(* CoDeSys 2.3.9.47 project: clv-199-wg-001.pro *)
(* Author: Diego Bernini *)
(* Libraries: SerComm.lib 31.5.11 08:54:36, SysLibEvent.lib 2.12.10 14:48:34, SysLibFile.lib 2.12.10 14:48:34, SysLibPlcCtrl.lib 2.12.10 14:48:32, SysLibRtc.lib 2.12.10 14:48:32, SysLibSockets.lib 10.2.11 09:20:54, 01_Lib_ClevergyUtils\ClevergyUtils_wg880_v2.lib 27.7.16 09:27:07, Util.lib 26.9.14 11:12:46, Visual.lib 2.12.10 14:48:34, WagoLibIdent.lib 25.2.13 11:12:16, WagoLibStatus.lib 2.12.10 14:48:32, Standard.lib 2.12.10 14:48:34, SYSLIBCALLBACK.LIB 2.12.10 14:48:32, mod_com.lib 2.12.10 14:48:32, MBus_03.lib 9.2.13 17:51:58, Modb_l05.lib 13.5.15 10:30:08, Serial_Interface_01.lib 22.4.13 12:50:14, WagoLibMBX_01.lib 20.3.12 16:32:40, WagoLibModbus_IP_01.lib 24.7.13 15:05:58, SysLibTime.lib 2.12.10 14:48:32 *)

(* PLC configuration (modules and I/O channels)
0750-1506 8DI / 8DO 24V DC 0.5A [Type_34_8_Channels] node 0, in %IB20 out %QB20 {INTTypePAAssignment = PLC; INTTypeModule = plugged}
  OUT2_VPN AT %IX10.0 [BOOLOnX_I] Ch_1 Digital input
  LAMP_AL AT %QX10.0 [BOOLOnX_Q] Ch_1 Digital output
  STATO_PORTA_QE AT %IX10.1 [BOOLOnX_I] Ch_2 Digital input
  AT %QX10.1 [BOOLOnX_Q] Ch_2 Digital output
  AT %IX10.2 [BOOLOnX_I] Ch_3 Digital input
  AT %QX10.2 [BOOLOnX_Q] Ch_3 Digital output
  AT %IX10.3 [BOOLOnX_I] Ch_4 Digital input
  AT %QX10.3 [BOOLOnX_Q] Ch_4 Digital output
  AT %IX10.4 [BOOLOnX_I] Ch_5 Digital input
  AT %QX10.4 [BOOLOnX_Q] Ch_5 Digital output
  AT %IX10.5 [BOOLOnX_I] Ch_6 Digital input
  AT %QX10.5 [BOOLOnX_Q] Ch_6 Digital output
  AT %IX10.6 [BOOLOnX_I] Ch_7 Digital input
  AT %QX10.6 [BOOLOnX_Q] Ch_7 Digital output
  AT %IX10.7 [BOOLOnX_I] Ch_8 Digital input
  AT %QX10.7 [BOOLOnX_Q] Ch_8 Digital output
AT %IB0 [BYTEOnB_I] First Byte of 8
AT %QB0 [BYTEOnB_Q] First Byte of 8
AT %IB8 [BYTEOnB_I] First Byte of 8
AT %QB8 [BYTEOnB_Q] First Byte of 8
0750-0650/0003-0000#03 RS 232 C Interface (Adjustable), 3 Byte [Type_21_1_Channels] node 3, in %IB24 out %QB24 {INTTypePAAssignment = PLC; INTTypeModule = plugged}
  AT %IX8.0 [BOOLOnX_I] Transmission acknowledgement
  AT %IX8.1 [BOOLOnX_I] Reception request
  AT %IX8.2 [BOOLOnX_I] Initialization acknowledgement
  AT %IX8.3 [BOOLOnX_I] Input buffer is full
  AT %IX8.4 [BOOLOnX_I] Number of received characters Bit 0
  AT %IX8.5 [BOOLOnX_I] Number of received characters Bit 1
  AT %IX8.6 [BOOLOnX_I] Number of received characters Bit 2
  AT %IB17 [BYTEOnB_I] Input data Byte 0
  AT %IB18 [BYTEOnB_I] Input data Byte 1
  AT %IB19 [BYTEOnB_I] Input data Byte 2
  AT %QX8.0 [BOOLOnX_Q] Transmission request
  AT %QX8.1 [BOOLOnX_Q] Reception acknowledgement
  AT %QX8.2 [BOOLOnX_Q] Initialization request
  AT %QX8.4 [BOOLOnX_Q] Number of characters Bit 0
  AT %QX8.5 [BOOLOnX_Q] Number of characters Bit 1
  AT %QX8.6 [BOOLOnX_Q] Number of characters Bit 2
  AT %QB17 [BYTEOnB_Q] Output data Byte 0
  AT %QB18 [BYTEOnB_Q] Output data Byte 1
  AT %QB19 [BYTEOnB_Q] Output data Byte 2
Fieldbus variables [FB_VARS] node 1, in %IB0 out %QB0
Flag variables [FLAG_VARS] node 2, in %IB0 out %QB0
Modbus-Master [MB_MASTER] node 3, in %IB0 out %QB0
*)

(* Global variable list: Global_Constants *)
VAR_GLOBAL CONSTANT

	Plant_NAME		: STRING :='cySN:199  cyVER:0 - Humanitas PIO X ';
	Plant_SN			: DWORD  :=199;  	         	(* S/N Impianto di telecontrollo *)
	Plant_SW_VER		: WORD   :=0;				(* Versione SW installata *)

	(* Plant-dependent constants *)
	(*Plant_ANZ_Frer			: BYTE	 :=24; *)
	Plant_ANZ_ABB		: BYTE	 :=19;
	(*Plant_GASM			: BYTE	 :=1; *)

	MODBUS_MAX_DEVICE	:BYTE:=19;
	MODBUS_MAX_REG 		: BYTE:=10;
	POLLING_TIME				:TIME:=T#10s;

	(* Filesystem *)
	FilesPath  		: STRING :='S:\';

	(* TCP Logger *)
	Logger_SERVER		: STRING:='';
	Logger_IP				: STRING:='192.168.100.3';
	Logger_PORT			: WORD  :=80;
	Logger_GETSTART		: STRING:='GET /cygmsrv/hsgm.ashx?';
	Logger_GETEND		: STRING:='$R$N$R$N';
	Logger_CHECK			: STRING:='True';
	Logger_CRLF			: STRING:='$R$N';
	Logger_DataFile			: STRING:='S:\LOG.DAT';
	Logger_DataFileOld		: STRING:='S:\LOG.BCK';
	Logger_IndexFile		: STRING:='S:\LOG.IDX';
	Logger_ConnRetries		: BYTE:=5;
	Logger_RecoverMsgs	: BYTE:=25;

	(* TCP Remote *)
	Remote_PORT			: WORD  :=10;
	Remote_WELCOME	: STRING:='Connected$R$N';
	Remote_OK				: STRING:='OK$R$N';
	Remote_ERROR		: STRING:='ERROR$R$N';

	(* TCP Sockets *)
	MAX_SEND_TCP_SERVER					 : DWORD:=6000;(*60000*)
	MAX_RECEIVE_TCP_SERVER				 : DWORD:=3000;
	MAX_RECEIVE_TCP_SERVER_SOCKET	  : DWORD:=1500;
	MAX_SEND_TCP_CLIENT					 : DWORD:=6000;(*15000*)
	MAX_RECEIVE_TCP_CLIENT				 : DWORD:=1500;
	MAX_RECEIVE_TCP_CLIENT_SOCKET		 : DWORD:=1500;
	MAX_RECEIVE_UDP_SERVER				 : INT  :=1472;
	MAX_RECEIVE_UDP_CLIENT				 : INT  :=1472;
	CONNECT_WATCHDOG_TIME				 : TIME :=t#10s;

	(* Colour defines *)
	COLOR_RED			: DWORD	:= 16#2020F0;
	COLOR_YELLOW		: DWORD	:= 16#20F0F0;
	COLOR_GREEN			: DWORD	:= 16#20F020;
	COLOR_GREEN_OFF		: DWORD := 16#006000;

END_VAR

(* Global variable list: Global_Variables *)
VAR_GLOBAL

	SYS    : typ_SYS;
	Logger : typ_Logger;

	Lamp	:	LAMP_AL_GENERALE; (* Per gestione allarme generico impianto *)

	MODB01 : obj_MODBUS	:= ( ID:=1 , (*COM:=2,*) BAUDRATE:=BAUD_9600, RS485:=TRUE, STOP_BITS:=STOPBITS_2,TIME_OUT_TIME:=t#1s);
	MODB02 : obj_MODBUS	:= ( ID:=2 , (*COM:=3,*) BAUDRATE:=BAUD_9600, RS485:=TRUE, STOP_BITS:=STOPBITS_2,TIME_OUT_TIME:=t#1s);
	ANZ_ABB				:	ARRAY[1..Plant_ANZ_ABB] OF obj_MODBUS_ABB_DMTME72;

	testANZ : ARRAY[1..19,1..23] OF REAL;

	MODBUS_RegDescr : ARRAY[1..MODBUS_MAX_DEVICE, 1..MODBUS_MAX_REG] OF STRING(20);
	MODBUS_RegAddress : ARRAY[1..MODBUS_MAX_DEVICE, 1..MODBUS_MAX_REG] OF WORD;
	MODBUS_RegQuantity : ARRAY[1..MODBUS_MAX_DEVICE, 1..MODBUS_MAX_REG] OF BYTE;
	MODBUS_RegValueType : ARRAY[1..MODBUS_MAX_DEVICE, 1..MODBUS_MAX_REG] OF en_Modbus_Reg_Type;


	MBUS01 : obj_MBUS							:= ( ID:=1 , COM:=4, BAUDRATE:=BAUD_2400 );
	CTB01  : obj_MBUS_CTB_SHARKY775			:= ( ID:=1 , ADDRESS:=16#58083647);
	CTB02  : obj_MBUS_CTB_SHARKY775			:= ( ID:=2 , ADDRESS:=16#56203308);
	CTB03  : obj_MBUS_CTB_SHARKY775			:= ( ID:=3 , ADDRESS:=16#58083750);
	CTB04  : obj_MBUS_CTB_SHARKY775			:= ( ID:=4 , ADDRESS:=16#58083646);
	CTB05  : obj_MBUS_CTB_SHARKY775			:= ( ID:=5 , ADDRESS:=16#56203321);
	CTB06  : obj_MBUS_CTB_SHARKY775			:= ( ID:=6 , ADDRESS:=16#58083749);
	CTB07  : obj_MBUS_CTB_SHARKY775			:= ( ID:=7 , ADDRESS:=16#56203320);
	CTB08  : obj_MBUS_CTB_SHARKY775			:= ( ID:=8 , ADDRESS:=16#58083751);
	CTB09  : obj_MBUS_CTB_SHARKY775			:= ( ID:=9 , ADDRESS:=16#55400970);
	CTB10  : obj_MBUS_CTB_SHARKY775			:= ( ID:=10 , ADDRESS:=16#55973781);

	testCTB : ARRAY[1..10,1..5] OF STRING(21);

	RichiestaLogDaRemoto: BOOL;

END_VAR

(* Data type *)
TYPE en_Modbus_Reg_Type :
(
	VALUE_REAL_SWAP		:=0,
	VALUE_REAL_NO_SWAP,
	VALUE_UINT ,
	VALUE_WORD,
	VALUE_DECIMAL_WORD_3,
	VALUE_32
);
END_TYPE

(* Data type *)
TYPE typ_GASM :
STRUCT
	Vb			: STRING;		(* HEX f64 m^3 *)
	Vm			: DWORD;		(* m^3 *)
	P			: REAL;		(* bar *)
	T			: REAL;		(* °C *)
	C			: REAL;
	Vbs			: STRING;		(* HEX F64 m^3 *)
	Vb_d_d		: STRING;		(* HEX F64 m^3 *)
	Vb_d_m		: STRING;		(* HEX F64 m^3 *)
	Vm_d_d		: DWORD;		(* m^3 *)
	Q			: REAL;		(* m^3/h *)
	Qb			: REAL;		(* m^3/h *)
	BC_EVC		: REAL;		(*E-1  % *)
	BV_EVC		: REAL;		(* V *)
	Status		: DWORD;		(* Status bits *)

END_STRUCT
END_TYPE

(* Data type *)
TYPE typ_GASMBASIC :
STRUCT
	Vb			: REAL;		(* m^3 *)
	Vm			: REAL;		(* m^3 *)
	P			: REAL;		(* bar *)
	T			: REAL;		(* °C *)
	C			: REAL;
	Q			: REAL;		(* m^3/h *)
	Qb			: REAL;		(* m^3/h *)
	BC_EVC		: REAL;		(*% *)
END_STRUCT
END_TYPE

(* Data type in Plant_Objects *)
TYPE typ_MODBUS_ABB_DMTME72 :
STRUCT
	V_3P		: DWORD; (* V *)
	V_L1N		: DWORD;
	V_L2N		: DWORD;
	V_L3N		: DWORD;
	V_L1L2		: DWORD;
	V_L2L3		: DWORD;
	V_L3L1		: DWORD;
	I_3P		: DWORD; (* 10^-3 A *)
	I_L1		: DWORD;
	I_L2		: DWORD;
	I_L3		: DWORD;
	PF_3P		: DINT;	 (* 10^-3 *)
	PF_L1		: DINT;
	PF_L2		: DINT;
	PF_L3		: DINT;
	COS_3P		: DINT;  (*NO!*)
	COS_L1		: DINT;
	COS_L2		: DINT;
	COS_L3		: DINT;
	VA_3P		: DWORD; (* VA *)(*NO!*)
	VA_L1		: DWORD;
	VA_L2		: DWORD;
	VA_L3		: DWORD;
	P_3P		: DWORD; (* W *)
	P_L1		: DWORD;
	P_L2		: DWORD;
	P_L3		: DWORD;
	Q_3P		: DWORD; (* VAr *)
	Q_L1		: DWORD;
	Q_L2		: DWORD;
	Q_L3		: DWORD;

	WH_3P		: DWORD; (* 10^-1 kWh *)
	VARH_3P		: DWORD; (* 10^-1 kVArh *)
	FREQ		: DWORD; (* 10^-3 Hz *)

	I_L1_Max	: DWORD;
	I_L2_Max	: DWORD;
	I_L3_Max	: DWORD;
	P_3P_Max	: DWORD;
	Q_3P_Max	: DWORD;
	P_3P_Avg15m	: DWORD;

END_STRUCT
END_TYPE

(* Data type in Plant_Objects *)
TYPE typ_MODBUS_ELGAS_MINIELCOR :
STRUCT
	Vb			: ARRAY [0..3] OF WORD;	(* m^3 *)
	Vm			: DWORD;				(* m^3 *)
	P			: REAL;					(* bar *)
	T			: REAL;					(* °C *)
	C			: REAL;
	Vbs			: ARRAY [0..3] OF WORD;	(* m^3 *)
	Vb_d_d		: ARRAY [0..3] OF WORD;	(* m^3 *)
	Vb_d_m		: ARRAY [0..3] OF WORD;	(* m^3 *)
	Vm_d_d		: DWORD;				(* m^3 *)
	Q			: REAL;					(* m^3/h *)
	Qb			: REAL;					(* m^3/h *)

	BC_EVC		: REAL;			(* % *)
	BV_EVC		: REAL;			(* V *)
	D_Err		: WORD;			(* 0:OK, 1:FAIL *)
	Status		: DWORD;		(* Status bits *)

END_STRUCT
END_TYPE

(* Data type *)
TYPE typ_MODBUS_ELSTER_EK220 :
STRUCT
	Vb			: REAL;	(* m^3 *)
	Vm			: REAL;				(* m^3 *)
	P			: REAL;					(* bar *)
	T			: REAL;					(* °C *)
	C			: REAL;
	Q			: REAL;					(* m^3/h *)
	Qb			: REAL;					(* m^3/h *)

	BC_EVC		: REAL;			(* % *)

END_STRUCT
END_TYPE

(* Data type in Plant_Objects *)
TYPE typ_MODBUS_FRER_QUBOH :
STRUCT
	V_L1N		:	DINT;	(* E-3 V *)
	V_L2N		:	DINT;
	V_L3N		:	DINT;
	V_L1L2		:	DINT;
	V_L2L3		:	DINT;
	V_L3L1		:	DINT;
	I_L1			:	DINT;	(* E-3 A *)
	I_L2			:	DINT;
	I_L3			:	DINT;

	FREQ		:	DWORD;	(* E-3 Hz *)

	P_3P			:	DINT;	(* W *)
	Q_3P		:	DINT;	(* VAr *)
	PF_3P		:	DINT;	(* E-3 *)
	WH_3P		:	DINT;	(* Wh *)
	VARH_3P		:	DINT;	(* VArh *)
	Multiplier	:	DWORD;

	V_3P		:	DINT;	(* E-3 V *)
	I_3P		:	DINT;	(* E-3 A *)

	COS_3P		:	DINT;	(* E-3 *)

	VA_3P		:	DINT;	(* VA *)
	P_L1		:	DWORD;	(* W *)
	P_L2		:	DWORD;
	P_L3		:	DWORD;
	Q_L1		:	DINT;	(* VAr *)
	Q_L2		:	DINT;
	Q_L3		:	DINT;
	VA_L1		:	DINT;	(* VA *)
	VA_L2		:	DINT;
	VA_L3		:	DINT;
	PF_L1		:	DINT;	(* E-3 *)
	PF_L2		:	DINT;
	PF_L3		:	DINT;
	COS_L1		:	DINT;	(* E-3 *)
	COS_L2		:	DINT;
	COS_L3		:	DINT;

	P_3P_Max	:	DINT;	(* W *)
	P_3P_Avg		:	DINT;

	I_L1_Max	:	DINT;	(* E-3 A *)
	I_L2_Max	:	DINT;
	I_L3_Max	:	DINT;

	Q_3P_Max	:	DINT;	(* VAr *)

END_STRUCT
END_TYPE

(* Data type in Plant_Objects *)
TYPE typ_MODBUS_VAR : (* Gestione parametri MODBUS *)
STRUCT
	SlaveAddress	: BYTE;
	FunCode			: BYTE;
	FunAddress		: WORD;
	Refresh_Time	: BYTE; (* 0:No refresh x:Refresh in seconds *)
	Refresh_Cnt		: BYTE; (* INTERNAL *)
	Variable		: POINTER TO ARRAY [0..124] OF WORD;	(* For classical ModBus it has to be equal to "typModbusResponse.Data"
																that is an array of 125 word ([0..124]) *)
	Variable_Size	: BYTE;
	Variable_Mirror : WORD; (* INTERNAL [Force refresh on read variables when <>0] *)
END_STRUCT
END_TYPE

(* POU PLC_PRG, ST *)
PROGRAM PLC_PRG
VAR
	Timer1: TON; (* Fast controls tick *)
	Timer2: TON; (* Plant control tick *)
	Timer3: TON; (* Logger timer *)

	i : INT;
	status : BYTE;
	eseguiLog:INT;
	Ton_pausaTrig: TON;


END_VAR
(******************************************************************************
 ****                           MAIN TASK CODE                             ****
 ******************************************************************************

	Network setup:
		IP  = 192.168.100.2 | MSK = 255.255.255.0
		GW	= 192.168.100.1 | DNS = 192.168.100.1
		SNTP = 193.204.114.232 (3600s) ==> 192.168.100.3

*)

(*==============================*)
(*===== Main status machine ====*)
(*==============================*)
Main_Stm();

(*==============================*)
(*== System cycle operations ===*)
(*==============================*)
(* Execute TCP processes *)
Logger_Proc();
Remote_Proc();

(* Execute Cron Editor commands *)
(*CronEd();*)

(**** SIMULATION ONLY ****)
(*...*)
(*
FOR i:=1 TO Plant_ANZ_Frer BY 1 DO
	testANZ[i,1]:=DINT_TO_REAL(ANZ_FRER[i].Data.V_L1N/1000);
	testANZ[i,2]:=DINT_TO_REAL(ANZ_FRER[i].Data.V_L2N/1000);
	testANZ[i,3]:=DINT_TO_REAL(ANZ_FRER[i].Data.V_L3N/1000);
	testANZ[i,4]:=DINT_TO_REAL(ANZ_FRER[i].Data.V_L1L2/1000);
	testANZ[i,5]:=DINT_TO_REAL(ANZ_FRER[i].Data.V_L2L3/1000);
	testANZ[i,6]:=DINT_TO_REAL(ANZ_FRER[i].Data.V_L3L1/1000);
	testANZ[i,7]:=DWORD_TO_REAL(ANZ_FRER[i].Data.FREQ);
	testANZ[i,8]:=DINT_TO_REAL(ANZ_FRER[i].Data.I_L1);
	testANZ[i,9]:=DINT_TO_REAL(ANZ_FRER[i].Data.I_L2);
	testANZ[i,10]:=DINT_TO_REAL(ANZ_FRER[i].Data.I_L3);
	testANZ[i,11]:=DINT_TO_REAL(ANZ_FRER[i].Data.I_L1_Max);
	testANZ[i,12]:=DINT_TO_REAL(ANZ_FRER[i].Data.I_L2_Max);
	testANZ[i,13]:=DINT_TO_REAL(ANZ_FRER[i].Data.I_L3_Max);
	testANZ[i,14]:=DINT_TO_REAL(ANZ_FRER[i].Data.PF_L1);
	testANZ[i,15]:=DINT_TO_REAL(ANZ_FRER[i].Data.PF_L2);
	testANZ[i,16]:=DINT_TO_REAL(ANZ_FRER[i].Data.PF_L3);
	testANZ[i,17]:=DINT_TO_REAL(ANZ_FRER[i].Data.P_3P);
	testANZ[i,18]:=DINT_TO_REAL(ANZ_FRER[i].Data.P_3P_Avg);
	testANZ[i,19]:=DINT_TO_REAL(ANZ_FRER[i].Data.P_3P_Max);
	testANZ[i,20]:=DINT_TO_REAL(ANZ_FRER[i].Data.Q_3P);
	testANZ[i,21]:=DINT_TO_REAL(ANZ_FRER[i].Data.Q_3P_Max);
	testANZ[i,22]:=DINT_TO_REAL(ANZ_FRER[i].Data.WH_3P);
	testANZ[i,23]:=DINT_TO_REAL(ANZ_FRER[i].Data.VARH_3P);
END_FOR
*)
FOR i:=1 TO Plant_ANZ_ABB BY 1 DO

	testANZ[i,1]:=DWORD_TO_REAL(ANZ_ABB[i].Data.V_L1N);
	testANZ[i,2]:=DWORD_TO_REAL(ANZ_ABB[i].Data.V_L2N);
	testANZ[i,3]:=DWORD_TO_REAL(ANZ_ABB[i].Data.V_L3N);
	testANZ[i,4]:=DWORD_TO_REAL(ANZ_ABB[i].Data.V_L1L2);
	testANZ[i,5]:=DWORD_TO_REAL(ANZ_ABB[i].Data.V_L2L3);
	testANZ[i,6]:=DWORD_TO_REAL(ANZ_ABB[i].Data.V_L3L1);
	testANZ[i,7]:=DWORD_TO_REAL(ANZ_ABB[i].Data.FREQ);
	testANZ[i,8]:=DWORD_TO_REAL(ANZ_ABB[i].Data.I_L1);
	testANZ[i,9]:=DWORD_TO_REAL(ANZ_ABB[i].Data.I_L2);
	testANZ[i,10]:=DWORD_TO_REAL(ANZ_ABB[i].Data.I_L3);
	testANZ[i,11]:=DWORD_TO_REAL(ANZ_ABB[i].Data.I_L1_Max);
	testANZ[i,12]:=DWORD_TO_REAL(ANZ_ABB[i].Data.I_L2_Max);
	testANZ[i,13]:=DWORD_TO_REAL(ANZ_ABB[i].Data.I_L3_Max);
	testANZ[i,14]:=DINT_TO_REAL(ANZ_ABB[i].Data.PF_L1);
	testANZ[i,15]:=DINT_TO_REAL(ANZ_ABB[i].Data.PF_L2);
	testANZ[i,16]:=DINT_TO_REAL(ANZ_ABB[i].Data.PF_L3);
	testANZ[i,17]:=DWORD_TO_REAL(ANZ_ABB[i].Data.P_3P);
	testANZ[i,18]:=DWORD_TO_REAL(ANZ_ABB[i].Data.P_3P_Avg15m);
	testANZ[i,19]:=DWORD_TO_REAL(ANZ_ABB[i].Data.P_3P_Max);
	testANZ[i,20]:=DWORD_TO_REAL(ANZ_ABB[i].Data.Q_3P);
	testANZ[i,21]:=DWORD_TO_REAL(ANZ_ABB[i].Data.Q_3P_Max);
	testANZ[i,22]:=DWORD_TO_REAL(ANZ_ABB[i].Data.WH_3P);
	testANZ[i,23]:=DWORD_TO_REAL(ANZ_ABB[i].Data.VARH_3P);
END_FOR

testCTB[1,1]:=CTB01.M1.utFTemp.Value;
testCTB[1,2]:=CTB01.M1.utRTemp.Value;
testCTB[1,3]:=CTB01.M1.utFlow.Value;
testCTB[1,4]:=CTB01.M1.utPower.Value;
testCTB[1,5]:=CTB01.M1.utEnergy.Value;

testCTB[2,1]:=CTB02.M1.utFTemp.Value;
testCTB[2,2]:=CTB02.M1.utRTemp.Value;
testCTB[2,3]:=CTB02.M1.utFlow.Value;
testCTB[2,4]:=CTB02.M1.utPower.Value;
testCTB[2,5]:=CTB02.M1.utEnergy.Value;

testCTB[3,1]:=CTB03.M1.utFTemp.Value;
testCTB[3,2]:=CTB03.M1.utRTemp.Value;
testCTB[3,3]:=CTB03.M1.utFlow.Value;
testCTB[3,4]:=CTB03.M1.utPower.Value;
testCTB[3,5]:=CTB03.M1.utEnergy.Value;

testCTB[4,1]:=CTB04.M1.utFTemp.Value;
testCTB[4,2]:=CTB04.M1.utRTemp.Value;
testCTB[4,3]:=CTB04.M1.utFlow.Value;
testCTB[4,4]:=CTB04.M1.utPower.Value;
testCTB[4,5]:=CTB04.M1.utEnergy.Value;

testCTB[5,1]:=CTB05.M1.utFTemp.Value;
testCTB[5,2]:=CTB05.M1.utRTemp.Value;
testCTB[5,3]:=CTB05.M1.utFlow.Value;
testCTB[5,4]:=CTB05.M1.utPower.Value;
testCTB[5,5]:=CTB05.M1.utEnergy.Value;

testCTB[6,1]:=CTB06.M1.utFTemp.Value;
testCTB[6,2]:=CTB06.M1.utRTemp.Value;
testCTB[6,3]:=CTB06.M1.utFlow.Value;
testCTB[6,4]:=CTB06.M1.utPower.Value;
testCTB[6,5]:=CTB06.M1.utEnergy.Value;

testCTB[7,1]:=CTB07.M1.utFTemp.Value;
testCTB[7,2]:=CTB07.M1.utRTemp.Value;
testCTB[7,3]:=CTB07.M1.utFlow.Value;
testCTB[7,4]:=CTB07.M1.utPower.Value;
testCTB[7,5]:=CTB07.M1.utEnergy.Value;

testCTB[8,1]:=CTB08.M1.utFTemp.Value;
testCTB[8,2]:=CTB08.M1.utRTemp.Value;
testCTB[8,3]:=CTB08.M1.utFlow.Value;
testCTB[8,4]:=CTB08.M1.utPower.Value;
testCTB[8,5]:=CTB08.M1.utEnergy.Value;

testCTB[9,1]:=CTB09.M1.utFTemp.Value;
testCTB[9,2]:=CTB09.M1.utRTemp.Value;
testCTB[9,3]:=CTB09.M1.utFlow.Value;
testCTB[9,4]:=CTB09.M1.utPower.Value;
testCTB[9,5]:=CTB09.M1.utEnergy.Value;

testCTB[10,1]:=CTB10.M1.utFTemp.Value;
testCTB[10,2]:=CTB10.M1.utRTemp.Value;
testCTB[10,3]:=CTB10.M1.utFlow.Value;
testCTB[10,4]:=CTB10.M1.utPower.Value;
testCTB[10,5]:=CTB10.M1.utEnergy.Value;

(*
FOR i:=1 TO Plant_GASM BY 1 DO
	testGASMBASIC[i,1]:=GASM[i].measures.Vb;
	testGASMBASIC[i,2]:=GASM[i].measures.Vm;
	testGASMBASIC[i,3]:=GASM[i].measures.P;
	testGASMBASIC[i,4]:=GASM[i].measures.T;
	testGASMBASIC[i,5]:=GASM[i].measures.C;
	testGASMBASIC[i,6]:=GASM[i].measures.Q;
	testGASMBASIC[i,7]:=GASM[i].measures.Qb;
	testGASMBASIC[i,7]:=GASM[i].measures.BC_EVC;
END_FOR
*)
END_PROGRAM
ACTION Main_Stm:
CASE Sys.Status OF

	S_STARTUP:
		Sys.Status:=S_INIT_RTC;

	S_INIT_RTC:
		(* Check RTC and update from network *)
		RTC_Update();
		(* Check time *)
		IF Sys.Time_Year>2000 THEN
			Sys.Status:=S_INIT_VAR;
		END_IF

	S_INIT_VAR:
		LogEv(EL_Wrn,EO_SYS,0,1,CONCAT('System_startup_v',WORD_TO_STRING(Plant_SW_VER)));

		(* Conditional settings for LUXs *)

	(*	FOR i:=1 TO Plant_ANZ_Frer BY 1 DO
			ANZ_Frer[i](ID:=INT_TO_BYTE(i), Address:=INT_TO_BYTE(i), ModBus:=MODB01);
		END_FOR
      
		FOR i:=1 TO Plant_ANZ_ABB BY 1 DO
			ANZ_ABB[i](ID:=Plant_ANZ_Frer+INT_TO_BYTE(i), Address:=Plant_ANZ_Frer+INT_TO_BYTE(i), ModBus:=MODB01);
		END_FOR
	*)
		FOR i:=1 TO 14 BY 1 DO
			ANZ_ABB[i](ID:=INT_TO_BYTE(i), Address:=INT_TO_BYTE(i), ModBus:=MODB01,COM:=2);
		END_FOR
		FOR i:=15 TO Plant_ANZ_ABB BY 1 DO
			ANZ_ABB[i](ID:=INT_TO_BYTE(i), Address:=INT_TO_BYTE(i-14), ModBus:=MODB02,COM:=3);
		END_FOR


		Sys.Status:=S_RUNNING;

	S_RUNNING:


		MODB01();
		FOR i:=1 TO 14 BY 1 DO
			ANZ_ABB[i](ModBus:=MODB01,Refresh_Period:=t#1m,COM:=2 );
		END_FOR


		MODB02();
		ANZ_ABB[15](ModBus:=MODB02,Refresh_Period:=t#1m,COM:=3 );

		FOR i:=15 TO Plant_ANZ_ABB BY 1 DO
			ANZ_ABB[i](ModBus:=MODB02,Refresh_Period:=t#1m,COM:=3 );
		END_FOR



		(* Execute MBUS01 process *)
		MBUS01();
		CTB01( MBUS:=MBUS01,Refresh_Period:=t#1m );
		CTB02( MBUS:=MBUS01,Refresh_Period:=t#1m );
		CTB03( MBUS:=MBUS01,Refresh_Period:=t#1m );
		CTB04( MBUS:=MBUS01,Refresh_Period:=t#1m );
		CTB05( MBUS:=MBUS01,Refresh_Period:=t#1m );
		CTB06( MBUS:=MBUS01,Refresh_Period:=t#1m );
		CTB07( MBUS:=MBUS01,Refresh_Period:=t#1m );
		CTB08( MBUS:=MBUS01,Refresh_Period:=t#1m );
		CTB09( MBUS:=MBUS01,Refresh_Period:=t#1m );
		CTB10( MBUS:=MBUS01,Refresh_Period:=t#1m );


		status :=0;


		FOR i:=1 TO Plant_ANZ_ABB BY 1 DO IF ANZ_ABB[i].Status_Log=1 THEN status :=1;  END_IF	END_FOR

		IF CTB01.Status_Log=1 THEN status :=1;  END_IF
		IF CTB02.Status_Log=1 THEN status :=1;  END_IF
		IF CTB03.Status_Log=1 THEN status :=1;  END_IF
		IF CTB04.Status_Log=1 THEN status :=1;  END_IF
		IF CTB05.Status_Log=1 THEN status :=1;  END_IF
		IF CTB06.Status_Log=1 THEN status :=1;  END_IF
		IF CTB07.Status_Log=1 THEN status :=1;  END_IF
		IF CTB08.Status_Log=1 THEN status :=1;  END_IF
		IF CTB09.Status_Log=1 THEN status :=1;  END_IF
		IF CTB10.Status_Log=1 THEN status :=1;  END_IF

		FOR i:=1 TO Plant_ANZ_ABB BY 1 DO IF ANZ_ABB[i].Status_Log=2 THEN status :=2;  END_IF	END_FOR

		IF CTB01.Status_Log=2 THEN status :=2;  END_IF
		IF CTB02.Status_Log=2 THEN status :=2;  END_IF
		IF CTB03.Status_Log=2 THEN status :=2;  END_IF
		IF CTB04.Status_Log=2 THEN status :=2;  END_IF
		IF CTB05.Status_Log=2 THEN status :=2;  END_IF
		IF CTB06.Status_Log=2 THEN status :=2;  END_IF
		IF CTB07.Status_Log=2 THEN status :=2;  END_IF
		IF CTB08.Status_Log=2 THEN status :=2;  END_IF
		IF CTB09.Status_Log=2 THEN status :=2;  END_IF
		IF CTB10.Status_Log=2 THEN status :=2;  END_IF

		Lamp( Allarme:=	(status=2),
			  Warning:=  (status=1),
			  SistemaInAllarme => Sys.Alarm,
			 SistemaWarning => Sys.Warning,
			 AllarmeLampada=>LAMP_AL
			 );

		Timer1(IN:=NOT Timer1.Q,PT:=T#50ms);
		IF Timer1.Q THEN
			(* Update meters *)
			SCA_Proc();
			(* Update system checks *)
			SYS_Proc();

		END_IF

		Timer2(IN:=NOT Timer2.Q,PT:=T#500ms);
		IF Timer2.Q THEN
			(* Read current date/time *)
			RTC_Update();
			(* Execute plant operations *)
			(* LUX cronos *)
		END_IF

		Timer3(IN:=NOT Timer3.Q,PT:=T#5m);
		IF Timer3.Q OR RichiestaLogDaRemoto  THEN

			EseguiLog:=10;
			RichiestaLogDaRemoto:=FALSE;
			(* Trig logger *)
			(* LogTrig(); *)
			(* Execute temporary CSV logger *)
			(*CSV_Log();*)
		END_IF

		CASE Eseguilog OF

			10 : 	Ton_pausaTrig(IN:=FALSE , PT:=t#5s , Q=> , ET=> );
					Logger_Head();

					FOR i:=1 TO 10 BY 1 DO
  						 ANZ_ABB[i].AddLogData(ModBus:=MODB01);
					END_FOR

					Logger_Send();
					RichiestaLogDaRemoto:=FALSE;
					EseguiLog:=20;

			20: Ton_pausaTrig(IN:=TRUE , PT:=t#5s , Q=> , ET=> );
					IF Ton_pausaTrig.Q THEN
						EseguiLog:=30;
					END_IF

			30 : 	Ton_pausaTrig(IN:=FALSE , PT:=t#5s , Q=> , ET=> );
					Logger_Head();

					FOR i:=11 TO 19 BY 1 DO
   						ANZ_ABB[i].AddLogData(ModBus:=MODB01);
					END_FOR

					Logger_Send();

					EseguiLog:=60;

			(*40: Ton_pausaTrig(IN:=TRUE , PT:=t#5s , Q=> , ET=> );
					IF Ton_pausaTrig.Q THEN
						EseguiLog:=50;
					END_IF

			50 : 	Ton_pausaTrig(IN:=FALSE , PT:=t#5s , Q=> , ET=> );
					Logger_Head();


					Logger_Send();*)

					EseguiLog:=60;
			(*10 : 	Ton_pausaTrig(IN:=FALSE , PT:=t#5s , Q=> , ET=> );
					Logger_Head();

						FOR i:=1 TO 14 BY 1 DO
							ANZ_ABB[i].AddLogData(ModBus:=MODB01,COM:=2);
						END_FOR

					Logger_Send();
					Logger_Head();

						FOR i:=15 TO Plant_ANZ_ABB BY 1 DO
							ANZ_ABB[i].AddLogData(ModBus:=MODB02,COM:=3);
					      END_FOR

					Logger_Send();

					EseguiLog:=60;*)
			60: Ton_pausaTrig(IN:=TRUE , PT:=t#5s , Q=> , ET=> );
					IF Ton_pausaTrig.Q THEN
						EseguiLog:=70;
					END_IF
			70 : 	Ton_pausaTrig(IN:=FALSE , PT:=t#5s , Q=> , ET=> );
					Logger_Head();

				CTB01.AddLogData( MBUS:=MBUS01 );
				CTB02.AddLogData( MBUS:=MBUS01 );
				CTB03.AddLogData( MBUS:=MBUS01 );
				CTB04.AddLogData( MBUS:=MBUS01 );
				CTB05.AddLogData( MBUS:=MBUS01 );
				CTB06.AddLogData( MBUS:=MBUS01 );
				CTB07.AddLogData( MBUS:=MBUS01 );
				CTB08.AddLogData( MBUS:=MBUS01 );
				CTB09.AddLogData( MBUS:=MBUS01 );
				CTB10.AddLogData( MBUS:=MBUS01 );

	(*			FOR i:=1 TO Plant_GASM BY 1 DO
							GASM[i].AddLogData();
				END_FOR
      *)
				Logger_Send();

				EseguiLog:=200;


			200: RichiestaLogDaRemoto:=FALSE;

	END_CASE

	S_SHUTDOWN:
		(* Stop sistema *)
		Sys.Status:=S_STARTUP;

	S_HALT:
		(* Aspetta uscita manuale *)
		Sys.Status:=S_STARTUP;

ELSE
	Sys.Status:=S_STARTUP;
END_CASE;
END_ACTION

(* POU TCP_Remote/Remote_Proc, ST *)
PROGRAM Remote_Proc
VAR
	s1:         	TCPSERVER;
	Enable: 		BOOL;
	Connected: 		BOOL;
	Error: 			DINT;

	TxData:			ARRAY [0..MAX_SEND_TCP_SERVER] OF BYTE;
	TxLen:			DINT;
	TxTrig:			BOOL;

	RxData:			ARRAY [0..MAX_RECEIVE_TCP_SERVER] OF BYTE;
	RxLen:			DINT;

	Status:			DINT;

	(* Command interpreter *)

	Cmd_Buf:		ARRAY [0..MAX_RECEIVE_TCP_SERVER] OF BYTE;
	Cmd_Buf_U16:	POINTER TO WORD;
	Cmd_Buf_INT:	POINTER TO INT;
	Cmd_BufLen:		WORD;
	Cmd_St:			WORD;

	Cmd_Obj:		WORD;
	Cmd_ObjIdx:		WORD;
	Cmd_C:			WORD;
	Cmd_R:			WORD;
	Cmd_CLen:		WORD;
	Cmd_RLen:		WORD;

	i : WORD;
	j : INT;
	s2 : STRING;

	(* per aggiornare la data e l'ora *)
	SetAnno: INT;
	SetMese: INT;
	SetGiorno: INT;
	SetOra: INT;
	SetMinuti: INT;
	SetSecondi: INT;

	Plant_SW_VER: BOOL;
         (* specific for lux *)
	x: INT;
	NewValueTimer : DWORD;

END_VAR
(*=== State machine ===*)
CASE Status OF
	0: (* Startup *)
		TxLen:=0; TxTrig:=FALSE;
		RxLen:=0;
		Enable:=TRUE;
		Status:=1;

	1: (* Wait incoming connection *)
		IF Connected THEN
			(* Log access *)(*
			LogEv(EL_Log,EO_VPN,1,5,'Remote');*)
			(* Send welcome message *)(*
			ADDSTRING(pTxData:=ADR(TxData), pString:=ADR(Remote_WELCOME), TxLen:=TxLen);
			TxTrig:=TRUE;*)
			(* Reset vars *)
			Cmd_BufLen:=0;
			Cmd_St:=0;
			Status:=2;
		END_IF
		IF Error>1 THEN
			Enable:=FALSE;
			Status:=0;
		END_IF

	2: (* Wait command *)
		IF RxLen>0 THEN
			(*=== Interpreter start ===*)
			IF Cmd_BufLen+(RxLen/2)>=MAX_RECEIVE_TCP_SERVER THEN
				(* ERROR *)
				Cmd_BufLen:=0;
			ELSE
				i:=HEXTORAW(pString:=ADR(RxData), StringLen:=DINT_TO_WORD(RxLen), pData:=ADR(Cmd_Buf[Cmd_BufLen]));
				Cmd_BufLen:=Cmd_BufLen+i;
			END_IF
			IF Cmd_BufLen>=8 THEN
				Cmd_Buf_U16:=ADR(Cmd_Buf[6]);
				IF Cmd_BufLen>=(8+Cmd_Buf_U16^) THEN
					Cmd_CLen:=Cmd_Buf_U16^;
					Cmd_Buf_U16:=ADR(Cmd_Buf[0]); Cmd_Obj:=Cmd_Buf_U16^;
					Cmd_Buf_U16:=ADR(Cmd_Buf[2]); Cmd_ObjIdx:=Cmd_Buf_U16^;
					Cmd_Buf_U16:=ADR(Cmd_Buf[4]); Cmd_C:=Cmd_Buf_U16^;
					(* Log command *)(*
					s2:='RCmd_';		s2:=CONCAT(s2,WORD_TO_STRING(Cmd_Obj));
					s2:=CONCAT(s2,'_'); s2:=CONCAT(s2,WORD_TO_STRING(Cmd_ObjIdx));
					s2:=CONCAT(s2,'_'); s2:=CONCAT(s2,WORD_TO_STRING(Cmd_C));
					s2:=CONCAT(s2,'_');	s2:=CONCAT(s2,WORD_TO_STRING(Cmd_CLen));
					LogEv(EL_Log,EO_VPN,1,6,s2);*)
					(* Execute command *)
					Command();
					Cmd_BufLen:=0;
				END_IF
			END_IF
			(*=== Interpreter end ===*)
			RxLen:=0;
		END_IF
		IF NOT Connected THEN
			Status:=0;
		END_IF

ELSE
	Status:=0;
END_CASE


(*=== Execute server lib ===*)
s1(
	xEnable				:= Enable,
	wPortNumber			:= Remote_PORT,
	tServerTimeOut		:= t#15m,
	ptSendData			:= ADR(TxData),
	diSendCount			:= TxLen,
	xStartSend			:= TxTrig,
	aReceiveBuffer		:= RxData,
	diReceiveCount		:= RxLen,
	xClientConnected	=> Connected,
	diError				=> Error
);
END_PROGRAM
ACTION Cmd_SYS:
(* Check index *)
IF Cmd_ObjIdx<>0 THEN
	Cmd_R:=2;
	RETURN;
END_IF

(* Process command *)
CASE Cmd_C OF

	0: (* ECHO *)
		IF Cmd_CLen<>0 THEN
			TxLen:=0;
		END_IF

	1: (* LOG REQUEST *)
		(*LogTrig();*)
		RichiestaLogDaRemoto:=TRUE;

	2: (* REARM *)
		Sys.Warning:=FALSE;
		Sys.Alarm:=FALSE;
		Sys.AlarmStop:=FALSE;

	3: (* GET INFO1 *)
		Cmd_RLen:=6;
		TxLen:=TxLen+RAWTOHEX(ADR(Plant_SN),4,ADR(TxData[TxLen]));
		TxLen:=TxLen+RAWTOHEX(ADR(Plant_SW_VER),2,ADR(TxData[TxLen]));

	14: (*  Imposto data e ora del PLC  *)


			Cmd_Buf_U16:=ADR(Cmd_Buf[8]);
			SetAnno:= Cmd_Buf_U16^; 												(* Anno *)
			Cmd_Buf_U16:=ADR(Cmd_Buf[10]);
			SetMese:= Cmd_Buf_U16^;												 	(* mese *)
			Cmd_Buf_U16:=ADR(Cmd_Buf[12]);
			SetGiorno:=( Cmd_Buf_U16^);											 	(* Giorno *)
			Cmd_Buf_U16:=ADR(Cmd_Buf[14]);
			SetOra:=( Cmd_Buf_U16^); 												(* ora *)
			Cmd_Buf_U16:=ADR(Cmd_Buf[16]);
			SetMinuti:= ( Cmd_Buf_U16^);										 	(* Minuti *)
			Cmd_Buf_U16:=ADR(Cmd_Buf[18]);
			SetSecondi:= ( Cmd_Buf_U16^);										 	(* secondi *)

			SysRtcSetTime((SetDataTime(SetAnno,SetMese,SetGiorno,SetOra,SetMinuti,SetSecondi)));

ELSE
	Cmd_R:=3;
END_CASE
END_ACTION
ACTION Command:
(* Default response OK/NODATA *)
Cmd_R:=0;
Cmd_RLen:=0;
TxLen:=16;

(* Check object *)
CASE Cmd_Obj OF

	EO_SYS:
		Cmd_SYS();

ELSE
	Cmd_R:=3;
END_CASE

(* Generate response *)
IF TxLen>0 THEN
	RAWTOHEX(ADR(Cmd_Obj)	,2,ADR(TxData[ 0]));
	RAWTOHEX(ADR(Cmd_ObjIdx),2,ADR(TxData[ 4]));
	RAWTOHEX(ADR(Cmd_R)		,2,ADR(TxData[ 8]));
	RAWTOHEX(ADR(Cmd_RLen)	,2,ADR(TxData[12]));
	TxTrig:=TRUE;
END_IF
END_ACTION

(* POU PLANT_PROCESS/SCA_Proc, ST *)
PROGRAM SCA_Proc
VAR
	(*SCA01_1	:	FLT_TAP;
	SCA01_2	:	FLT_TAP;
	SCA01_3	:	FLT_TAP;

	upd		:	BOOL;*)
END_VAR
(***** SCA01 *****)
(*SCA01_1(IN:=SCA01_1_DI);
IF SCA01_1.EVL THEN LogEv(EL_Wrn,EO_SCA,1,1,'1'); upd:=TRUE; END_IF
IF SCA01_1.EVH THEN	LogEv(EL_Log,EO_SCA,1,2,'1'); upd:=TRUE; END_IF

SCA01_2(IN:=SCA01_2_DI);
IF SCA01_2.EVL THEN	LogEv(EL_Wrn,EO_SCA,1,1,'2'); upd:=TRUE; END_IF
IF SCA01_2.EVH THEN	LogEv(EL_Log,EO_SCA,1,2,'2'); upd:=TRUE; END_IF

SCA01_3(IN:=SCA01_3_DI);
IF SCA01_3.EVL THEN	LogEv(EL_Wrn,EO_SCA,1,1,'3'); upd:=TRUE; END_IF
IF SCA01_3.EVH THEN	LogEv(EL_Log,EO_SCA,1,2,'3'); upd:=TRUE; END_IF

IF upd THEN
	upd:=FALSE;
	Logger_Head();
	AddLogData();
	Logger_Send();
END_IF*)
;
END_PROGRAM
ACTION AddLogData:
(*Logger.s1:='&SCA01=';
Logger.s1:=CONCAT(Logger.s1,BYTE_TO_STRING(BOOL_TO_BYTE(SCA01_1.OUT))		); Logger.s1:=CONCAT(Logger.s1,';');
Logger.s1:=CONCAT(Logger.s1,BYTE_TO_STRING(BOOL_TO_BYTE(SCA01_2.OUT))		); Logger.s1:=CONCAT(Logger.s1,';');
Logger.s1:=CONCAT(Logger.s1,BYTE_TO_STRING(BOOL_TO_BYTE(SCA01_3.OUT))		);
ADDSTRING(ADR(Logger.TData), ADR(Logger.s1), Logger.TLen);*)
;
END_ACTION

(* POU PLANT_PROCESS/SYS_Proc, ST *)
PROGRAM SYS_Proc
VAR

	fVPN		:FLT_TAP;  (* stato VPN*)
	fDoor		:FLT_TAP;  (* stato QE*)

END_VAR
(*### VPN Status Check ###*)
fVPN(IN:=OUT2_VPN);
IF fVPN.EVH THEN
	LogEv(EL_Log,EO_VPN,1,3,'STATUS_UP');
END_IF
IF fVPN.EVL THEN
	LogEv(EL_Wrn,EO_VPN,1,4,'STATUS_DOWN');
END_IF

(*### QE ###*)
fDoor(IN:=STATO_PORTA_QE);
IF fDoor.EVH THEN
	LogEv(EL_Log,EO_DOOR,1,1,'BOX_CLOSED');
END_IF
IF fDoor.EVL THEN
	LogEv(EL_Wrn,EO_DOOR,1,2,'BOX_OPENED');
END_IF
END_PROGRAM

(* POU ClevergyBlocks/BUILD_REAL_COPY, ST *)
FUNCTION BUILD_REAL_COPY : REAL
VAR_INPUT
		W1	:	WORD;
		W2	:	WORD;
END_VAR
VAR
 	awWords      : ARRAY[1..2] OF WORD;
  	pReal : POINTER TO REAL;
  	rReal : REAL;
END_VAR
awWords[1] := W1;
awWords[2] := W2;
pReal := ADR(awWords);
rReal := pReal^;
BUILD_REAL_COPY:=rReal;
END_FUNCTION

(* POU Plant_Objects/obj_MBUS, ST *)
FUNCTION_BLOCK obj_MBUS
(* === M-BUS PROTOCOL INTERFACE ===
   v1.0[16/03/05] - Added interface errors
*)
VAR_INPUT
	(* Settings *)
	ID				: BYTE;
	COM				: BYTE;
	BAUDRATE		: COM_BAUDRATE;
	(* Interface *)
	MBus 			: typMBus;
	MBus_Master 	: FbMBusMaster;
END_VAR
VAR_OUTPUT
	(* Status *)
	Status_Log		: BYTE;
	Status_Vis 		: DWORD;
END_VAR
VAR
	Alarm			: FLT_EVENT;
END_VAR
MBus_Master( bCOMPORT:=COM , enumBAUDRATE:=BAUDRATE , utMBus:=MBus );

(* Check status *)
Alarm(IN:=(MBus.bCOM_ERROR<>0));
IF Alarm.EVH THEN
	LogEv(EL_Alarm,EO_MBUS,ID,1,BYTE_TO_STRING(MBus.bCOM_ERROR));
END_IF
IF Alarm.EVL THEN
	LogEv(EL_Log,EO_MBUS,ID,2,'MBUS_OK');
END_IF

(* Log/visu status *)
   IF Alarm.IN   					THEN Status_Log:=2; Status_Vis:=16#2020F0;
ELSIF (MBus.bL1_ERROR AND 16#1F)<>0 THEN Status_Log:=1; Status_Vis:=16#20F0F0;
  				 					ELSE Status_Log:=0; Status_Vis:=16#20F020;
END_IF
END_FUNCTION_BLOCK

(* POU Plant_Objects/obj_MBUS_CTB_SHARKY775, ST *)
FUNCTION_BLOCK obj_MBUS_CTB_SHARKY775
(* === M-BUS CONTABILIZER SHARKY 775 ===
   v1.0[16/03/05] - Error management
*)
VAR_INPUT
	(* Settings *)
	ID				: BYTE;
	ADDRESS			: DWORD;
	Refresh_Period	: TIME:=t#3m;
	(* Controls *)
	Refresh_Auto	: BOOL:=TRUE; (* Enable automatic refresh *)
	Refresh_Now		: BOOL; 	  (* Force an immediate refresh *)
END_VAR
VAR_IN_OUT
	(* Interface *)
	MBUS			: obj_MBUS;
END_VAR
VAR_OUTPUT
	M1				: FbMBus_Heat;
	(* Status *)
	Status_Log		: BYTE;
	Status_Vis 		: DWORD;
END_VAR
VAR
	dly 	 	: TON := (PT:=t#5s);
	M1_Start	: BOOL;

	init_st		: BOOL;
	bus_st0		: BYTE;
	dev_st0		: BYTE;

(*	S1			: FbMBusSend;
	S1_Start	: BOOL;*)
(*	C1			: FbUnitConverter; *)
END_VAR
(* Auto refresh timer *)
dly(IN:=NOT (dly.Q OR Refresh_Now OR (NOT Refresh_Auto)));
(* Trigger refresh *)
IF dly.Q OR Refresh_Now THEN
	dly.PT:=Refresh_Period;
	Refresh_Now:=FALSE;
	(* Start reading *)
	M1.dwAdr:= ADDRESS;
	M1.xSND_NKE:=TRUE;
	M1_Start:=TRUE;
END_IF

(* Contabilizer module *)
M1(	utMBus:=MBUS.MBus, xStart:=M1_Start );

(* Extra actions *)
(*C1( utMBus:=MBUS.MBus, xStart:=C1_Start );*)

(* Check status *)
IF NOT init_st OR M1.bError<>bus_st0 OR M1.utMBInfo.bMStatus<>dev_st0 THEN
	init_st:=TRUE;
	bus_st0:=M1.bError; dev_st0:=M1.utMBInfo.bMStatus;
	IF bus_st0<>0 THEN
		LogEv(EL_Alarm,EO_CTB,ID,2,BYTE_TO_STRING(bus_st0));
		Status_Log:=2; Status_Vis:=16#2020F0;
	ELSE
		IF dev_st0<>0 THEN
			Status_Log:=2; Status_Vis:=16#2020F0;
			CASE dev_st0 OF
				16#08: LogEv(EL_Alarm,EO_CTB,ID,10,'C-1');
				16#04: LogEv(EL_Alarm,EO_CTB,ID,10,'E-8');
				16#28: LogEv(EL_Alarm,EO_CTB,ID,10,'E-4');
				16#50: LogEv(EL_Alarm,EO_CTB,ID,10,'E-1');
				16#70: LogEv(EL_Alarm,EO_CTB,ID,10,'E-7');
				16#84: LogEv(EL_Alarm,EO_CTB,ID,10,'E-9');
				16#B0: LogEv(EL_Wrn  ,EO_CTB,ID,10,'E-3');
				16#D0: LogEv(EL_Wrn  ,EO_CTB,ID,10,'E-6');
				16#F0: LogEv(EL_Alarm,EO_CTB,ID,10,'Leak');
				16#10: LogEv(EL_Wrn  ,EO_CTB,ID,10,'E-5'); Status_Log:=1; Status_Vis:=16#20F0F0;
			ELSE
				LogEv(EL_Alarm,EO_CTB,ID,10,BYTE_TO_STRING(dev_st0));
			END_CASE
		ELSE
			Status_Log:=0; Status_Vis:=16#20F020;
			LogEv(EL_Log,EO_CTB,ID,1,'');
		END_IF
	END_IF
END_IF
END_FUNCTION_BLOCK
ACTION AddLogData:
Logger.s1:=INSERT('&CTB=',BYTE_TO_STRING(ID),4);
IF ID<10 THEN Logger.s1:=INSERT(Logger.s1,'0',4); END_IF

Logger.s1:=CONCAT(Logger.s1,SEL(M1.utFTemp.Value='',M1.utFTemp.Value,'0'));		Logger.s1:=CONCAT(Logger.s1,';');
Logger.s1:=CONCAT(Logger.s1,SEL(M1.utRTemp.Value='',M1.utRTemp.Value,'0'));		Logger.s1:=CONCAT(Logger.s1,';');
Logger.s1:=CONCAT(Logger.s1,SEL(M1.utFlow.Value='',M1.utFlow.Value,'0'));		Logger.s1:=CONCAT(Logger.s1,';');
Logger.s1:=CONCAT(Logger.s1,SEL(M1.utPower.Value='',M1.utPower.Value,'0'));		Logger.s1:=CONCAT(Logger.s1,';');
Logger.s1:=CONCAT(Logger.s1,SEL(M1.utEnergy.Value='',M1.utEnergy.Value,'0'));		Logger.s1:=CONCAT(Logger.s1,';');

Logger.s1:=CONCAT(Logger.s1,BYTE_TO_STRING(Status_Log));
ADDSTRING(ADR(Logger.TData), ADR(Logger.s1), Logger.TLen);
END_ACTION

(* POU ClevergyBlocks/obj_MODBUS, ST *)
FUNCTION_BLOCK obj_MODBUS
(* === MODBUS PROTOCOL INTERFACE ===
   v1.1[19/06/15] - Added new VARS allocation and searching
*)
VAR CONSTANT
	VARS_Max	: BYTE := 32;
END_VAR
VAR_INPUT
	(* Settings *)
	ID			: BYTE;
	COM			: BYTE;
	BAUDRATE	: COM_BAUDRATE;
	RS485		: BOOL := FALSE;
	PARITY : COM_PARITY:=PARITY_NO;
	BIT_SIZE: COM_BYTESIZE:=BS_8;
	STOP_BITS :COM_STOPBITS:=STOPBITS_2;
	TIME_OUT_TIME : TIME:=t#250ms;

	(* Interface *)
	MB_MASTER	: MODBUS_EXTENDED_MASTER;
	MB_Start	: BOOL;
	MB_Query	: typModbusExtendedQuery;
	MB_Resp		: typModbusResponse;
	MB_Lock		: BOOL;
	MB_Obj		: en_SYS_Objects;
	MB_ObjId	: BYTE;

	(* Variables management *)
	VARS_En		: BOOL := FALSE;
	VARS		: ARRAY [0..VARS_Max] OF typ_MODBUS_VAR;
	VARS_Check	: BOOL;
	VARS_Alarm	: BOOL;

	(* Variables allocation *)
	VAR_Pointer : POINTER TO ARRAY[0..99] OF WORD;
	VAR_Cfg		: POINTER TO typ_MODBUS_VAR;
END_VAR
VAR_OUTPUT
	(* Status *)
	Status_Log	: BYTE;
	Status_Vis	: DWORD;
END_VAR
VAR
	sta         : BYTE :=0;
	i			: BYTE;
	j			: BYTE;

	AlarmCOM	: FLT_EVENT;	(* Physical error relative to serial port -> COM	*)
	AlarmMDB	: FLT_EVENT;	(* ModBus error due to communication protocol error	*)

	VarTmr		: TON := (PT:=T#1s);
	VarSta		: BYTE; (* Status *)
	VarCnt		: BYTE; (* Scan counter *)
	VarRetry	: BYTE;
	VarAlarm	: BYTE; (* Last variable with errors *)
END_VAR
MB_MASTER(ENABLE:=TRUE,	ASCII_Mode:=FALSE, bCOM_PORT:=COM, cbCOM_BAUDRATE:=BAUDRATE, cpCOM_PARITY:=PARITY ,
		csCOM_STOPBITS:=STOP_BITS ,	cbsCOM_BYTESIZE:=BIT_SIZE, cfCOM_FLOW_CONTROL:=SEL(RS485,NO_FLOW_CONTROL,HALFDUPLEX),
		tTIME_OUT:=TIME_OUT_TIME,	StartFunction:=MB_Start, ExtQuery:=MB_Query, Response:=MB_Resp);

(* Process variable management *)
IF VARS_En THEN VARS_Process(); END_IF

(* Check status *)
AlarmCOM(IN:=(MB_MASTER.bInterfaceError<>0));
IF AlarmCOM.EVH THEN
	LogEv(SEL(MB_MASTER.bInterfaceError<>3,EL_Wrn,EL_Alarm),EO_MODBUS,ID,1,BYTE_TO_STRING(MB_MASTER.bInterfaceError));
END_IF
IF AlarmCOM.EVL THEN								(* Trigger a fall edge: MODBUS back working *)
	LogEv(EL_Log,EO_MODBUS,ID,2,'MODBUS_OK');
END_IF

(* If VARS not active check if a protocol error has occured (if VARS active this check is already done in "VARS_Process"	*)
IF NOT VARS_En THEN

	AlarmMDB(IN:=(MB_MASTER.MB_Error<>0));
(*	IF AlarmMDB.EVH THEN
		LogEv(EL_Wrn,EO_MODBUS,ID,2,INT_TO_STRING(MB_MASTER.MB_Error));
	END_IF
	IF AlarmMDB.EVL THEN								(* Trigger a fall edge: MODBUS back working *)
		LogEv(EL_Log,EO_MODBUS,ID,2,'MODBUS_OK');
	END_IF
*)
END_IF

(* Log/visu status *)
IF AlarmCOM.IN THEN Status_Log:=2; Status_Vis:=COLOR_RED;
ELSIF Vars_Alarm OR AlarmMDB.IN THEN Status_Log:=1; Status_Vis:=COLOR_YELLOW;
ELSE Status_Log:=0; Status_Vis:=COLOR_GREEN;
END_IF
END_FUNCTION_BLOCK
ACTION VAR_Search:
(* Search VAR with specific pointer if not found return first free VAR
	[Last VAR is not active... used as safe area...] 
*)
j:=VARS_Max;
FOR i := 0 TO VARS_Max-1 DO
	IF VARS[i].Variable=0 AND j>i THEN j:=i; END_IF
	IF VARS[i].Variable=VAR_Pointer THEN
		VAR_Cfg:=ADR(VARS[i]);
		RETURN;
	END_IF
END_FOR
VAR_Cfg:=ADR(VARS[j]);
END_ACTION
ACTION VARS_Process:
(* Update var timers *)
VarTmr(IN:=(NOT VarTmr.Q));
IF VarTmr.Q THEN
	FOR i := 0 TO VARS_Max DO
		IF VARS[i].Refresh_Cnt>0 THEN VARS[i].Refresh_Cnt:=VARS[i].Refresh_Cnt-1; END_IF
	END_FOR
	VARS_Check:=TRUE;
END_IF


(* Process status *)
CASE VarSta OF
	0: (* === Init *)
		VarCnt:=0;
		VarSta:=1;

	1: (* === Wait check signal *)
		IF VARS_Check THEN				(* Decremented "Refresh_Cnt" *)
			VARS_Check:=FALSE;
			VarCnt:=0;
			VarSta:=2;
		END_IF

	2: (* === Check loop *)
		IF NOT (MB_Lock OR MB_Start) THEN
			WHILE VarCnt<=(VARS_Max-1) AND VarSta=2 DO
				(* Check only active vars *)
				IF VARS[VarCnt].Variable<>0 THEN			(* "Variable" is a pointer to word, so if 0 no address *)
					(* Check var auto-refresh on timer checks *)
					IF VARS[VarCnt].Refresh_Time>0 AND VARS[VarCnt].Refresh_Cnt=0 THEN
						VARS[VarCnt].Refresh_Cnt:=VARS[VarCnt].Refresh_Time;
						VarSta:=3;
					END_IF
					(* Check refresh for change or request *)
					CASE VARS[VarCnt].FunCode OF
						5,6,15,16: (* Write functions *)
							IF VARS[VarCnt].Variable_Size=1 THEN
								IF VARS[VarCnt].Variable^[0]<>VARS[VarCnt].Variable_Mirror THEN
									VARS[VarCnt].Variable_Mirror:=VARS[VarCnt].Variable^[0];
									VarSta:=3;
								END_IF
							ELSE
								IF VARS[VarCnt].Variable_Mirror<>0 THEN
									VARS[VarCnt].Variable_Mirror:=0;
									VarSta:=3;
								END_IF
							END_IF
						1,2,3,4: (* Read functions *)
							IF VARS[VarCnt].Variable_Mirror<>0 THEN
								VARS[VarCnt].Variable_Mirror:=0;
								VarSta:=3;
							END_IF
					END_CASE
				END_IF
				(* Process query *)
				IF VarSta=3 THEN
					MB_Lock:=TRUE;
					MB_Query.SlaveAddress:=VARS[VarCnt].SlaveAddress;
					MB_Query.FunctionCode:=VARS[VarCnt].FunCode;
					CASE VARS[VarCnt].FunCode OF
						16#5,16#6,16#F,16#10:
							MB_Query.Read_Quantity:=0;
							MB_Query.Read_StartAddress:=0;
							MB_Query.Write_StartAddress:=VARS[VarCnt].FunAddress;
							MB_Query.Write_Quantity:=VARS[VarCnt].Variable_Size;
							IF VARS[VarCnt].Variable_Size=200 THEN
								COPY_32SWAP16(VARS[VarCnt].Variable, ADR(MB_Query.Write_Data[0]));
							ELSIF VARS[VarCnt].Variable_Size>1 THEN
								MEMCPY(VARS[VarCnt].Variable, ADR(MB_Query.Write_Data[0]), 2*VARS[VarCnt].Variable_Size);
							ELSE
								MB_Query.Write_Data[0]:=VARS[VarCnt].Variable^[0];
							END_IF
						16#1,16#2,16#3,16#4:
							MB_Query.Read_StartAddress:=VARS[VarCnt].FunAddress;
							IF VARS[VarCnt].Variable_Size=200 THEN MB_Query.Read_Quantity:=2; ELSE
							  MB_Query.Read_Quantity:=VARS[VarCnt].Variable_Size;
							END_IF
							MB_Query.Write_StartAddress:=0;
							MB_Query.Write_Quantity:=0;
					END_CASE
					VarRetry:=0;
					MB_Start:=TRUE;
				ELSE
					VarCnt:=VarCnt+1;
				END_IF
			END_WHILE
			(* Check loop completed -> no actions *)
			IF VarSta=2 THEN VarSta:=1; END_IF
		END_IF

	3: (* === Wait & process MB response *)
		IF NOT MB_Start THEN
			IF MB_MASTER.MB_Error=0 THEN
				CASE VARS[VarCnt].FunCode OF
					1,2,3,4:
						IF VARS[VarCnt].Variable_Size=200 THEN
							COPY_32SWAP16(ADR(MB_Resp.Data), VARS[VarCnt].Variable);
						ELSIF VARS[VarCnt].Variable_Size>1 THEN
							MEMCPY(ADR(MB_Resp.Data), VARS[VarCnt].Variable, 2*VARS[VarCnt].Variable_Size);
						ELSE
							VARS[VarCnt].Variable^[0]:=MB_Resp.Data[0];
						END_IF
				END_CASE
				MB_Lock:=FALSE;
				(* Signal error recovery *)
				IF VARS_Alarm=TRUE AND VarCnt=VarAlarm THEN
					LogEv(EL_Wrn,EO_MODBUS,ID,5,'');
					VARS_Alarm:=FALSE;
				END_IF
				(* Next var *)
				VarCnt:=VarCnt+1;
				VarSta:=2;
			ELSE
				IF VarRetry<3 THEN
					VarRetry:=VarRetry+1;
					MB_Start:=TRUE;
				ELSE
					MB_Lock:=FALSE;
					(* Signal error *)
					IF VARS_Alarm=FALSE THEN
						LogEv(EL_Wrn,EO_MODBUS,ID,3,INT_TO_STRING(MB_MASTER.MB_Error));
						VARS_Alarm:=TRUE;
						VarAlarm:=VarCnt-1;
					END_IF
					(* Next var *)
					VarCnt:=VarCnt+1;
					VarSta:=2;
				END_IF
			END_IF
		END_IF

ELSE
	VarSta:=0;
END_CASE
END_ACTION

(* POU Plant_Objects/obj_MODBUS_ABB_DMTME72, ST *)
FUNCTION_BLOCK obj_MODBUS_ABB_DMTME72
VAR_INPUT
	(* Settings *)
	ID				: BYTE;
	ADDRESS			: BYTE:=31;
	Refresh_Period	: TIME:=t#1m;
	(* Controls *)
	Refresh_Auto	: BOOL:=TRUE; (* Enable automatic refresh *)
	Refresh_Now		: BOOL; 	  (* Force an immediate refresh *)
	COM			: BYTE;

END_VAR
VAR_IN_OUT
	MODBUS			: obj_MODBUS;
END_VAR
VAR_OUTPUT
	Data			: typ_MODBUS_ABB_DMTME72;
	(* Status *)
	Status_Log		: BYTE;
	Status_Vis 		: DWORD;
END_VAR
VAR
	dly 	 : TON := (PT:=t#5s);
	sta		 : BYTE; 	(* Status *)
	retry		: 	BYTE;


END_VAR
CASE sta OF
	0: (* === Wait update signals *)
		dly(IN:=NOT (dly.Q OR Refresh_Now OR (NOT Refresh_Auto)));
		IF dly.Q OR Refresh_Now THEN
			dly.PT:=Refresh_Period;
			Refresh_Now:=FALSE;
			sta:=1;
		END_IF

	1: (* === Start update when MB is free *)
		IF NOT (MODBUS.MB_Lock OR MODBUS.MB_Start) THEN
			MODBUS.COM:=COM;
			MODBUS.MB_Lock:=TRUE;
			MODBUS.MB_Query.SlaveAddress:=ADDRESS;
			MODBUS.MB_Query.FunctionCode:=16#03;
			(* Start query *)
			MODBUS.MB_Query.Read_StartAddress:=16#1000;
			MODBUS.MB_Query.Read_Quantity:=16#16;
			MODBUS.MB_Start:=TRUE;
			sta:=2;
		END_IF

	2:	IF NOT MODBUS.MB_Start THEN
			IF MODBUS.MB_MASTER.MB_Error<>MB_NO_ERROR OR MODBUS.MB_Resp.Error<>0 THEN
				sta:=100;
			ELSE
				(* Read response data *)
				COPY_32SWAP16(ADR(MODBUS.MB_Resp.Data[ 0]),ADR(Data.V_3P));
				COPY_32SWAP16(ADR(MODBUS.MB_Resp.Data[ 2]),ADR(Data.V_L1N));
				COPY_32SWAP16(ADR(MODBUS.MB_Resp.Data[ 4]),ADR(Data.V_L2N));
				COPY_32SWAP16(ADR(MODBUS.MB_Resp.Data[ 6]),ADR(Data.V_L3N));
				COPY_32SWAP16(ADR(MODBUS.MB_Resp.Data[ 8]),ADR(Data.V_L1L2));
				COPY_32SWAP16(ADR(MODBUS.MB_Resp.Data[10]),ADR(Data.V_L2L3));
				COPY_32SWAP16(ADR(MODBUS.MB_Resp.Data[12]),ADR(Data.V_L3L1));
				COPY_32SWAP16(ADR(MODBUS.MB_Resp.Data[14]),ADR(Data.I_3P));
				COPY_32SWAP16(ADR(MODBUS.MB_Resp.Data[16]),ADR(Data.I_L1));
				COPY_32SWAP16(ADR(MODBUS.MB_Resp.Data[18]),ADR(Data.I_L2));
				COPY_32SWAP16(ADR(MODBUS.MB_Resp.Data[20]),ADR(Data.I_L3));
				(* Start query *)
				MODBUS.MB_Query.Read_StartAddress:=16#1016;
				MODBUS.MB_Query.Read_Quantity:=16#10;
				MODBUS.MB_Start:=TRUE;
				sta:=3;
			END_IF
		END_IF

	3:	IF NOT MODBUS.MB_Start THEN
			IF MODBUS.MB_MASTER.MB_Error<>MB_NO_ERROR OR MODBUS.MB_Resp.Error<>0 THEN
				sta:=100;
			ELSE
				(* Read response data *)
				COPY_32SWAP16(ADR(MODBUS.MB_Resp.Data[ 0]),ADR(Data.PF_3P));
				COPY_32SWAP16(ADR(MODBUS.MB_Resp.Data[ 2]),ADR(Data.PF_L1));
				COPY_32SWAP16(ADR(MODBUS.MB_Resp.Data[ 4]),ADR(Data.PF_L2));
				COPY_32SWAP16(ADR(MODBUS.MB_Resp.Data[ 6]),ADR(Data.PF_L3));
				COPY_32SWAP16(ADR(MODBUS.MB_Resp.Data[ 8]),ADR(Data.COS_3P));
				COPY_32SWAP16(ADR(MODBUS.MB_Resp.Data[10]),ADR(Data.COS_L1));
				COPY_32SWAP16(ADR(MODBUS.MB_Resp.Data[12]),ADR(Data.COS_L2));
				COPY_32SWAP16(ADR(MODBUS.MB_Resp.Data[14]),ADR(Data.COS_L3));
				(* Start query *)
				MODBUS.MB_Query.Read_StartAddress:=16#1026;
				MODBUS.MB_Query.Read_Quantity:=16#10;
				MODBUS.MB_Start:=TRUE;
				sta:=5;
			END_IF
		END_IF

	5:	IF NOT MODBUS.MB_Start THEN
			IF MODBUS.MB_MASTER.MB_Error<>MB_NO_ERROR OR MODBUS.MB_Resp.Error<>0 THEN
				sta:=100;
			ELSE
				(* Read response data *)
				COPY_32SWAP16(ADR(MODBUS.MB_Resp.Data[ 0]),ADR(Data.VA_3P));
				COPY_32SWAP16(ADR(MODBUS.MB_Resp.Data[ 2]),ADR(Data.VA_L1));
				COPY_32SWAP16(ADR(MODBUS.MB_Resp.Data[ 4]),ADR(Data.VA_L2));
				COPY_32SWAP16(ADR(MODBUS.MB_Resp.Data[ 6]),ADR(Data.VA_L3));
				COPY_32SWAP16(ADR(MODBUS.MB_Resp.Data[ 8]),ADR(Data.P_3P));
				COPY_32SWAP16(ADR(MODBUS.MB_Resp.Data[10]),ADR(Data.P_L1));
				COPY_32SWAP16(ADR(MODBUS.MB_Resp.Data[12]),ADR(Data.P_L2));
				COPY_32SWAP16(ADR(MODBUS.MB_Resp.Data[14]),ADR(Data.P_L3));
				(* Start query *)
				MODBUS.MB_Query.Read_StartAddress:=16#1036;
				MODBUS.MB_Query.Read_Quantity:=16#0C;
				MODBUS.MB_Start:=TRUE;
				sta:=6;
			END_IF
		END_IF

	6:	IF NOT MODBUS.MB_Start THEN
			IF MODBUS.MB_MASTER.MB_Error<>MB_NO_ERROR OR MODBUS.MB_Resp.Error<>0 THEN
				sta:=100;
			ELSE
				(* Read response data *)
				COPY_32SWAP16(ADR(MODBUS.MB_Resp.Data[ 0]),ADR(Data.Q_3P));
				COPY_32SWAP16(ADR(MODBUS.MB_Resp.Data[ 2]),ADR(Data.Q_L1));
				COPY_32SWAP16(ADR(MODBUS.MB_Resp.Data[ 4]),ADR(Data.Q_L2));
				COPY_32SWAP16(ADR(MODBUS.MB_Resp.Data[ 6]),ADR(Data.Q_L3));
				COPY_32SWAP16(ADR(MODBUS.MB_Resp.Data[ 8]),ADR(Data.WH_3P));
				COPY_32SWAP16(ADR(MODBUS.MB_Resp.Data[10]),ADR(Data.VARH_3P));
				(* Start query *)
				MODBUS.MB_Query.Read_StartAddress:=16#1046;
				MODBUS.MB_Query.Read_Quantity:=16#02;
				MODBUS.MB_Start:=TRUE;
				sta:=7;
			END_IF
		END_IF

	7:	IF NOT MODBUS.MB_Start THEN
			IF MODBUS.MB_MASTER.MB_Error<>MB_NO_ERROR OR MODBUS.MB_Resp.Error<>0 THEN
				sta:=100;
			ELSE
				(* Read response data *)
				COPY_32SWAP16(ADR(MODBUS.MB_Resp.Data[ 0]),ADR(Data.FREQ));
				(* Start query *)
				MODBUS.MB_Query.Read_StartAddress:=16#1060;
				MODBUS.MB_Query.Read_Quantity:=16#0A;
				MODBUS.MB_Start:=TRUE;
				sta:=8;
			END_IF
		END_IF

	8:	IF NOT MODBUS.MB_Start THEN
			IF MODBUS.MB_MASTER.MB_Error<>MB_NO_ERROR OR MODBUS.MB_Resp.Error<>0 THEN
				sta:=100;
			ELSE
				(* Read response data *)
				COPY_32SWAP16(ADR(MODBUS.MB_Resp.Data[ 0]),ADR(Data.I_L1_Max));
				COPY_32SWAP16(ADR(MODBUS.MB_Resp.Data[ 2]),ADR(Data.I_L2_Max));
				COPY_32SWAP16(ADR(MODBUS.MB_Resp.Data[ 4]),ADR(Data.I_L3_Max));
				COPY_32SWAP16(ADR(MODBUS.MB_Resp.Data[ 6]),ADR(Data.P_3P_Max));
				COPY_32SWAP16(ADR(MODBUS.MB_Resp.Data[ 8]),ADR(Data.Q_3P_Max));
				(* Start query *)
				MODBUS.MB_Query.Read_StartAddress:=16#1070;
				MODBUS.MB_Query.Read_Quantity:=16#02;
				MODBUS.MB_Start:=TRUE;
				sta:=9;
			END_IF
		END_IF

	9:	IF NOT MODBUS.MB_Start THEN
			IF MODBUS.MB_MASTER.MB_Error<>MB_NO_ERROR OR MODBUS.MB_Resp.Error<>0 THEN
				sta:=100;
			ELSE
				(* Read response data *)
				COPY_32SWAP16(ADR(MODBUS.MB_Resp.Data[ 0]),ADR(Data.P_3P_Avg15m));
				(* Release MODBUS *)
				MODBUS.MB_Lock:=FALSE;
				(* Update status *)
				Status_Log:=0;
				Status_Vis:=16#20F020;
				sta:=0;
			END_IF
		END_IF

	100: (* === Check MODBUS error *)

		MODBUS.MB_Lock:=FALSE;

			(* Retries *)
			retry:=retry+1;

			IF retry>3 THEN
				retry:=0;
				(* Signal event *)
				IF Status_Log<>2 THEN
					LogEv(EL_Alarm,EO_ANZ,ID,2,SEL(ModBus.MB_MASTER.MB_Error<>0,'0','1'));
				END_IF
				(* Update status *)
				Status_Log:=2;
			END_IF

			sta := 0;

ELSE
	sta:=0;
END_CASE

IF Status_Log=2 THEN Status_Vis := COLOR_RED;
ELSE Status_Vis := COLOR_GREEN;
END_IF
END_FUNCTION_BLOCK
ACTION AddLogData:
Logger.s1:=INSERT('&ANZ=',BYTE_TO_STRING(ID),4);
IF ID<10 THEN Logger.s1:=INSERT(Logger.s1,'0',4); END_IF

Logger.s1:=CONCAT(Logger.s1,DWORD_TO_STRING(Data.V_L1N));		Logger.s1:=CONCAT(Logger.s1,';');
Logger.s1:=CONCAT(Logger.s1,DWORD_TO_STRING(Data.V_L2N));		Logger.s1:=CONCAT(Logger.s1,';');
Logger.s1:=CONCAT(Logger.s1,DWORD_TO_STRING(Data.V_L3N));		Logger.s1:=CONCAT(Logger.s1,';');
Logger.s1:=CONCAT(Logger.s1,DWORD_TO_STRING(Data.V_L1L2));		Logger.s1:=CONCAT(Logger.s1,';');
Logger.s1:=CONCAT(Logger.s1,DWORD_TO_STRING(Data.V_L2L3));		Logger.s1:=CONCAT(Logger.s1,';');
Logger.s1:=CONCAT(Logger.s1,DWORD_TO_STRING(Data.V_L3L1));		Logger.s1:=CONCAT(Logger.s1,';');
Logger.s1:=CONCAT(Logger.s1,DWORD_TO_STRING(Data.FREQ));		Logger.s1:=CONCAT(Logger.s1,';');

Logger.s1:=CONCAT(Logger.s1,DWORD_TO_STRING(Data.I_L1));		Logger.s1:=CONCAT(Logger.s1,';');
Logger.s1:=CONCAT(Logger.s1,DWORD_TO_STRING(Data.I_L2));		Logger.s1:=CONCAT(Logger.s1,';');
Logger.s1:=CONCAT(Logger.s1,DWORD_TO_STRING(Data.I_L3));		Logger.s1:=CONCAT(Logger.s1,';');
Logger.s1:=CONCAT(Logger.s1,DWORD_TO_STRING(Data.I_L1_Max)); 	Logger.s1:=CONCAT(Logger.s1,';');
Logger.s1:=CONCAT(Logger.s1,DWORD_TO_STRING(Data.I_L2_Max)); 	Logger.s1:=CONCAT(Logger.s1,';');
Logger.s1:=CONCAT(Logger.s1,DWORD_TO_STRING(Data.I_L3_Max)); 	Logger.s1:=CONCAT(Logger.s1,';');

Logger.s1:=CONCAT(Logger.s1,DINT_TO_STRING(Data.PF_L1));		Logger.s1:=CONCAT(Logger.s1,';');
Logger.s1:=CONCAT(Logger.s1,DINT_TO_STRING(Data.PF_L2));		Logger.s1:=CONCAT(Logger.s1,';');
Logger.s1:=CONCAT(Logger.s1,DINT_TO_STRING(Data.PF_L3));		Logger.s1:=CONCAT(Logger.s1,';');

Logger.s1:=CONCAT(Logger.s1,DWORD_TO_STRING(Data.P_3P));		Logger.s1:=CONCAT(Logger.s1,';');
Logger.s1:=CONCAT(Logger.s1,DWORD_TO_STRING(Data.P_3P_Avg15m)); Logger.s1:=CONCAT(Logger.s1,';');
Logger.s1:=CONCAT(Logger.s1,DWORD_TO_STRING(Data.P_3P_Max)); 	Logger.s1:=CONCAT(Logger.s1,';');

Logger.s1:=CONCAT(Logger.s1,DWORD_TO_STRING(Data.Q_3P));		Logger.s1:=CONCAT(Logger.s1,';');
Logger.s1:=CONCAT(Logger.s1,DWORD_TO_STRING(Data.Q_3P_Max));	Logger.s1:=CONCAT(Logger.s1,';');

Logger.s1:=CONCAT(Logger.s1,DWORD_TO_STRING(Data.WH_3P));		Logger.s1:=CONCAT(Logger.s1,';');
Logger.s1:=CONCAT(Logger.s1,DWORD_TO_STRING(Data.VARH_3P));		Logger.s1:=CONCAT(Logger.s1,';');

Logger.s1:=CONCAT(Logger.s1,BYTE_TO_STRING(Status_Log));
ADDSTRING(ADR(Logger.TData), ADR(Logger.s1), Logger.TLen);
END_ACTION

(* POU PLANTCONFIG/Plant_LogTrig, ST *)
FUNCTION Plant_LogTrig : BOOL
VAR_INPUT
END_VAR
VAR
	i:INT;
END_VAR
;
END_FUNCTION

(* POU Utils Functions/RAW16TOHEXSTR, ST *)
FUNCTION RAW16TOHEXSTR : STRING(128)
VAR_INPUT
	pData: POINTER TO BYTE;
	DataLen: BYTE;
END_VAR
VAR
	pt: POINTER TO BYTE;
	xl: BYTE;
END_VAR
pt:=ADR(RAW16TOHEXSTR);
xl:=0;

WHILE DataLen>0 AND xl<120 DO

	pData:=pData+1;

	pt^ := (pData^ / 16#10) + 48 + (((pData^ / 16#10)/10)*7);
	pt:=pt+1;
	pt^ := (pData^ AND 16#0F)  + 48 + (((pData^ AND 16#0F)/10)*7);
	pt:=pt+1;

	pData:=pData-1;

	pt^ := (pData^ / 16#10) + 48 + (((pData^ / 16#10)/10)*7);
	pt:=pt+1;
	pt^ := (pData^ AND 16#0F)  + 48 + (((pData^ AND 16#0F)/10)*7);
	pt:=pt+1;

	xl:=xl+4;

	DataLen:=DataLen-2;
	pData:=pData+2;

END_WHILE

pt^:=0;
END_FUNCTION

(* POU ClevergyBlocks/REAL_TO_DOUBLE_HEX_STRING, ST *)
FUNCTION REAL_TO_DOUBLE_HEX_STRING : STRING
VAR_INPUT
 NUM:REAL;
END_VAR
VAR
END_VAR
REAL_TO_DOUBLE_HEX_STRING:='CIA0';
END_FUNCTION

(* Visualisation PLC_VISU
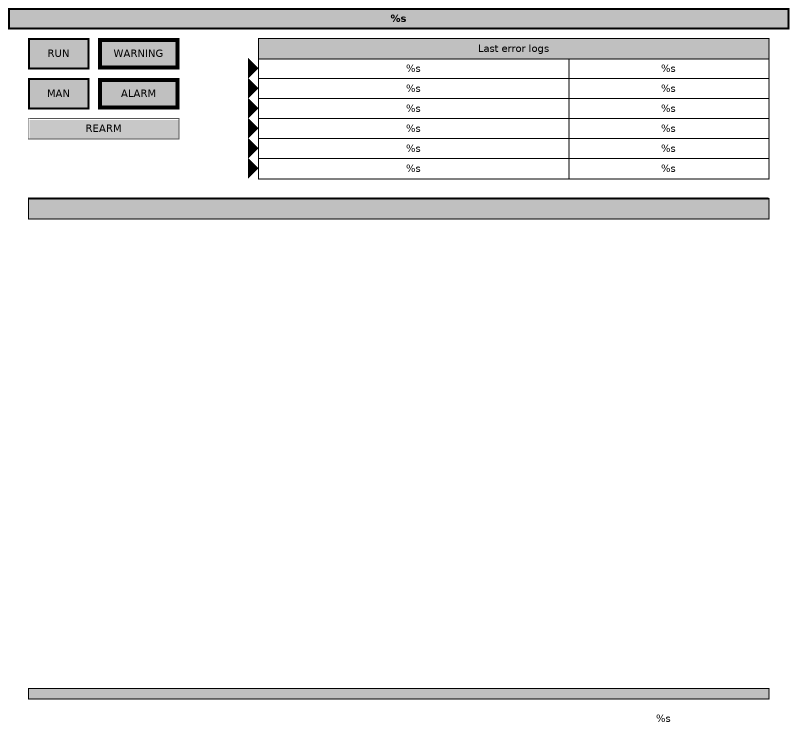
rectangle at (10,0)-(791,21): text "%s"; shows .Plant_NAME
rounded rectangle at (30,30)-(91,61): text "RUN"; alarm colour if NOT Mode_Manual; runs INTERN ASSIGN Mode_Manual:=(FALSE)
rounded rectangle at (30,70)-(91,101): text "MAN"; alarm colour if Mode_Manual; runs INTERN ASSIGN Mode_Manual:=(TRUE)
rectangle at (570,50)-(771,71): text "%s"; shows Sys.LastLogs_Msg[0]
polygon at (250,150)-(260,170): invisible if Sys.LastLogs_Idx<>0
rectangle at (570,70)-(771,91): text "%s"; shows Sys.LastLogs_Msg[1]
polygon at (250,50)-(260,70): invisible if Sys.LastLogs_Idx<>1
rectangle at (570,90)-(771,111): text "%s"; shows Sys.LastLogs_Msg[2]
polygon at (250,70)-(260,90): invisible if Sys.LastLogs_Idx<>2
rectangle at (570,110)-(771,131): text "%s"; shows Sys.LastLogs_Msg[3]
polygon at (250,90)-(260,110): invisible if Sys.LastLogs_Idx<>3
rectangle at (570,130)-(771,151): text "%s"; shows Sys.LastLogs_Msg[4]
polygon at (250,110)-(260,130): invisible if Sys.LastLogs_Idx<>4
rectangle at (570,150)-(771,171): text "%s"; shows Sys.LastLogs_Msg[5]
polygon at (250,130)-(260,150): invisible if Sys.LastLogs_Idx<>5
rectangle at (260,50)-(571,71): text "%s"; shows Sys.LastLogs_Dat[0]
rectangle at (260,70)-(571,91): text "%s"; shows Sys.LastLogs_Dat[1]
rectangle at (260,90)-(571,111): text "%s"; shows Sys.LastLogs_Dat[2]
rectangle at (260,110)-(571,131): text "%s"; shows Sys.LastLogs_Dat[3]
rectangle at (260,130)-(571,151): text "%s"; shows Sys.LastLogs_Dat[4]
rectangle at (260,150)-(571,171): text "%s"; shows Sys.LastLogs_Dat[5]
rectangle at (100,70)-(181,101): text "ALARM"; alarm colour if Sys.Alarm; runs INTERN ASSIGN Mode_Manual:=(FALSE)
rectangle at (100,30)-(181,61): text "WARNING"; alarm colour if Sys.Warning; runs INTERN ASSIGN Mode_Manual:=(TRUE)
button at (30,110)-(181,131): text "REARM"; runs INTERN ASSIGN Sys.Alarm:=(FALSE);INTERN ASSIGN Sys.Warning:=(FALSE)
rectangle at (260,30)-(771,51): text "Last error logs"
rectangle at (560,700)-(771,721): text "%s"; shows Sys.Time_LogString
3 more shapes without text or variables
4 elements of other kinds (tables, trends, ...) not read
*)

(* Visualisation PLC_VISU_ANZ
1 elements of other kinds (tables, trends, ...) not read
*)

(* Visualisation PLC_VISU_CTB_GASM
1 elements of other kinds (tables, trends, ...) not read
*)
